(*
    Tests the free function F_AnyToUnionValue.
*)
{attribute 'call_after_init'}
FUNCTION_BLOCK FB_AnyToUnionValue_Test EXTENDS TcUnit.FB_TestSuite IMPLEMENTS TcUnit.I_RunnableTestSuite
VAR
    Assert : TcUnit.FB_Assert;
    
    aBit : BIT := 1; // Only structures and function blocks can have BIT defined
END_VAR

METHOD FB_init : BOOL
VAR_INPUT
	bInitRetains : BOOL; // if TRUE, the retain variables are initialized (warm start / cold start)
	bInCopyCode : BOOL;  // if TRUE, the instance afterwards gets moved into the copy code (online change)
END_VAR
SUPER^.RegisterTestSuite(THIS^);
END_METHOD

METHOD RunTests : TCUNIT.E_TestSuiteRunState
Test_BOOL();
Test_BIT();
Test_BYTE();
Test_WORD();
Test_DWORD();
Test_LWORD();
Test_SINT();
Test_INT();
Test_DINT();
Test_LINT();
Test_USINT();
Test_UINT();
Test_UDINT();
Test_ULINT();
Test_REAL();
Test_LREAL();
Test_STRING();
Test_STRING_2();
Test_WSTRING();
Test_TIME();
Test_DATE();
Test_DATE_AND_TIME();
Test_TIME_OF_DAY();
Test_LTIME();

RunTests := TCUNIT.E_TestSuiteRunState.FINISHED;
END_METHOD

METHOD PRIVATE Test_BIT
VAR
    result : U_ExpectedOrActual;
END_VAR
TEST('Test_BIT');

result := TcUnit.F_AnyToUnionValue(AnyValue := aBit);

Assert.AssertEquals(Expected := aBit,
                    Actual := result.bitExpectedOrActual,
                    Message := 'Values differ');
END_METHOD

METHOD PRIVATE Test_BOOL
VAR
    a : BOOL := TRUE;
    result : U_ExpectedOrActual;
END_VAR
TEST('Test_BOOL');

result := TcUnit.F_AnyToUnionValue(AnyValue := a);

Assert.AssertEquals(Expected := a,
                    Actual := result.boolExpectedOrActual,
                    Message := 'Values differ');
END_METHOD

METHOD PRIVATE Test_BYTE
VAR
    a : BYTE := 16#8A;
    result : U_ExpectedOrActual;
END_VAR
TEST('Test_BYTE');

result := TcUnit.F_AnyToUnionValue(AnyValue := a);

Assert.AssertEquals(Expected := a,
                    Actual := result.byteExpectedOrActual,
                    Message := 'Values differ');
END_METHOD

METHOD PRIVATE Test_DATE
VAR
    a : DATE := D#2106-02-05;
    result : U_ExpectedOrActual;
END_VAR
TEST('Test_DATE');

result := TcUnit.F_AnyToUnionValue(AnyValue := a);

Assert.AssertEquals(Expected := a,
                    Actual := result.dateExpectedOrActual,
                    Message := 'Values differ');
END_METHOD

METHOD PRIVATE Test_DATE_AND_TIME
VAR
    a : DATE_AND_TIME := DT#2106-02-06-06:28:15;
    result : U_ExpectedOrActual;
END_VAR
TEST('Test_DATE_AND_TIME');

result := TcUnit.F_AnyToUnionValue(AnyValue := a);

Assert.AssertEquals(Expected := a,
                    Actual := result.dateandtimeExpectedOrActual,
                    Message := 'Values differ');
END_METHOD

METHOD PRIVATE Test_DINT
VAR
    a : DINT := 143251;
    result : U_ExpectedOrActual;
END_VAR
TEST('Test_DINT');

result := TcUnit.F_AnyToUnionValue(AnyValue := a);

Assert.AssertEquals(Expected := a,
                    Actual := result.dintExpectedOrActual,
                    Message := 'Values differ');
END_METHOD

METHOD PRIVATE Test_DWORD
VAR
    a : DWORD := 16#3456CDEF;
    result : U_ExpectedOrActual;
END_VAR
TEST('Test_DWORD');

result := TcUnit.F_AnyToUnionValue(AnyValue := a);

Assert.AssertEquals(Expected := a,
                    Actual := result.dwordExpectedOrActual,
                    Message := 'Values differ');
END_METHOD

METHOD PRIVATE Test_INT
VAR
    a : INT := -32000;
    result : U_ExpectedOrActual;
END_VAR
TEST('Test_INT');

result := TcUnit.F_AnyToUnionValue(AnyValue := a);

Assert.AssertEquals(Expected := a,
                    Actual := result.intExpectedOrActual,
                    Message := 'Values differ');
END_METHOD

METHOD PRIVATE Test_LINT
VAR
    a : LINT := -31243145;
    result : U_ExpectedOrActual;
END_VAR
TEST('Test_LINT');

result := TcUnit.F_AnyToUnionValue(AnyValue := a);

Assert.AssertEquals(Expected := a,
                    Actual := result.lintExpectedOrActual,
                    Message := 'Values differ');
END_METHOD

METHOD PRIVATE Test_LREAL
VAR
    a : LREAL := 43123923124.745423;
    result : U_ExpectedOrActual;
END_VAR
TEST('Test_LREAL');

result := TcUnit.F_AnyToUnionValue(AnyValue := a);

Assert.AssertEquals(Expected := a,
                    Actual := result.lrealExpectedOrActual,
                    Message := 'Values differ');
END_METHOD

METHOD PRIVATE Test_LTIME
VAR
    a : LTIME := LTIME#213502D23H34M33S709MS551US615NS;
    result : U_ExpectedOrActual;
END_VAR
TEST('Test_LTIME');

result := TcUnit.F_AnyToUnionValue(AnyValue := a);

Assert.AssertEquals(Expected := a,
                    Actual := result.ltimeExpectedOrActual,
                    Message := 'Values differ');
END_METHOD

METHOD PRIVATE Test_LWORD
VAR
    a : LWORD := 16#456CDEF987654321;
    result : U_ExpectedOrActual;
END_VAR
TEST('Test_LWORD');

result := TcUnit.F_AnyToUnionValue(AnyValue := a);

Assert.AssertEquals(Expected := a,
                    Actual := result.lwordExpectedOrActual,
                    Message := 'Values differ');
END_METHOD

METHOD PRIVATE Test_REAL
VAR
    a : REAL := 431239.423;
    result : U_ExpectedOrActual;
END_VAR
TEST('Test_REAL');

result := TcUnit.F_AnyToUnionValue(AnyValue := a);

Assert.AssertEquals(Expected := a,
                    Actual := result.realExpectedOrActual,
                    Message := 'Values differ');
END_METHOD

METHOD PRIVATE Test_SINT
VAR
    a : SINT := 100;
    result : U_ExpectedOrActual;
END_VAR
TEST('Test_SINT');

result := TcUnit.F_AnyToUnionValue(AnyValue := a);

Assert.AssertEquals(Expected := a,
                    Actual := result.sintExpectedOrActual,
                    Message := 'Values differ');
END_METHOD

METHOD PRIVATE Test_STRING
VAR
    a : STRING := 'This is a random string';
    result : U_ExpectedOrActual;
END_VAR
TEST('Test_STRING');

result := TcUnit.F_AnyToUnionValue(AnyValue := a);

Assert.AssertEquals(Expected := a,
                    Actual := result.stringExpectedOrActual,
                    Message := 'Values differ');
END_METHOD

METHOD PRIVATE Test_STRING_2
VAR
    a : Tc2_System.T_MaxString := '8YNn5KOmPC4dAcpOBdLWnw4WkN126EwXsj65xeurG48gWBepinNaOIKeCVMtWNBSxQWPdtUYiAusDkjMLtQhDtiWbwvmoKcFwiUGDd7pOe0fd52J7hK60oaYAX6VWWmceLJX8utaDVrVzCGXafeZLeHl6jj5enfjg4tfb2WMEBdsBuG2iDKwzwhBLCPqXDnhe5HbemIbtZT7p62OEj2oDqiIYDD6tZdlhBCCelDBx6dbIp32wFm0TpRKsTiwkZ6'; // 255 characters
    result : U_ExpectedOrActual;
END_VAR
TEST('Test_STRING_2');

result := TcUnit.F_AnyToUnionValue(AnyValue := a);

Assert.AssertEquals(Expected := a,
                    Actual := result.stringExpectedOrActual,
                    Message := 'Values differ');
END_METHOD

METHOD PRIVATE Test_TIME
VAR
    a : TIME := T#15M20S;
    result : U_ExpectedOrActual;
END_VAR
TEST('Test_TIME');

result := TcUnit.F_AnyToUnionValue(AnyValue := a);

Assert.AssertEquals(Expected := a,
                    Actual := result.timeExpectedOrActual,
                    Message := 'Values differ');
END_METHOD

METHOD PRIVATE Test_TIME_OF_DAY
VAR
    a : TIME_OF_DAY := TOD#15:36:30.123;
    result : U_ExpectedOrActual;
END_VAR
TEST('Test_TIME_OF_DAY');

result := TcUnit.F_AnyToUnionValue(AnyValue := a);

Assert.AssertEquals(Expected := a,
                    Actual := result.timeofdayExpectedOrActual,
                    Message := 'Values differ');
END_METHOD

METHOD PRIVATE Test_UDINT
VAR
    a : UDINT := 2555;
    result : U_ExpectedOrActual;
END_VAR
TEST('Test_UDINT');

result := TcUnit.F_AnyToUnionValue(AnyValue := a);

Assert.AssertEquals(Expected := a,
                    Actual := result.udintExpectedOrActual,
                    Message := 'Values differ');
END_METHOD

METHOD PRIVATE Test_UINT
VAR
    a : UINT := 34523;
    result : U_ExpectedOrActual;
END_VAR
TEST('Test_UINT');

result := TcUnit.F_AnyToUnionValue(AnyValue := a);

Assert.AssertEquals(Expected := a,
                    Actual := result.uintExpectedOrActual,
                    Message := 'Values differ');
END_METHOD

METHOD PRIVATE Test_ULINT
VAR
    a : ULINT := 25555423;
    result : U_ExpectedOrActual;
END_VAR
TEST('TEST_ULINT');

result := TcUnit.F_AnyToUnionValue(AnyValue := a);

Assert.AssertEquals(Expected := a,
                    Actual := result.ulintExpectedOrActual,
                    Message := 'Values differ');
END_METHOD

METHOD PRIVATE Test_USINT
VAR
    a : USINT := 255;
    result : U_ExpectedOrActual;
END_VAR
TEST('Test_USINT');

result := TcUnit.F_AnyToUnionValue(AnyValue := a);

Assert.AssertEquals(Expected := a,
                    Actual := result.usintExpectedOrActual,
                    Message := 'Values differ');
END_METHOD

METHOD PRIVATE Test_WORD
VAR
    a : WORD := 16#ABCD;
    result : U_ExpectedOrActual;
END_VAR
TEST('Test_WORD');

result := TcUnit.F_AnyToUnionValue(AnyValue := a);

Assert.AssertEquals(Expected := a,
                    Actual := result.wordExpectedOrActual,
                    Message := 'Values differ');
END_METHOD

METHOD PRIVATE Test_WSTRING
VAR
    a : WSTRING := "This is a random string";
    result : U_ExpectedOrActual;
END_VAR
TEST('Test_WSTRING');

result := TcUnit.F_AnyToUnionValue(AnyValue := a);

Assert.AssertEquals(Expected := a,
                    Actual := result.wstringExpectedOrActual,
                    Message := 'Values differ');
END_METHOD

END_FUNCTION_BLOCK

(* stored: Version 1.1.0.1, ProductVersion 3.1.4022.16
   POU FB_AnyToUnionValue_Test: Id {0cc46357-158c-41b7-afc0-2c79ec82f0f6}, SpecialFunc None
   Method FB_init: Id {0485650c-1465-4486-a734-95b061eb38ae}
   Method RunTests: Id {7fda42d2-1918-424a-ba0f-a586afc09af2}
   Method Test_BIT: Id {2bab70c5-093e-48a7-94e6-ae7f2bb2e7b3}
   Method Test_BOOL: Id {48f55beb-9fc1-4336-8784-72fc7eda80de}
   Method Test_BYTE: Id {226781dc-3660-487a-bcbd-00cc36750e0e}
   Method Test_DATE: Id {84a5fde1-b357-4804-bf01-5c83bfeb54b3}
   Method Test_DATE_AND_TIME: Id {76b46507-8743-481c-8853-3b45d1544ad5}
   Method Test_DINT: Id {c81a9536-5ff4-4424-9f7e-1d8c5133b5e3}
   Method Test_DWORD: Id {e6dfcf37-a491-45b2-9543-b7fdd8847283}
   Method Test_INT: Id {77ff5bf1-1822-4366-a4ee-34a185c0d47e}
   Method Test_LINT: Id {d2a7cc80-d43e-4823-a346-11defa0d180f}
   Method Test_LREAL: Id {af2fee48-9d46-49ec-9fe0-6a046d6c2f7d}
   Method Test_LTIME: Id {1affac86-d501-40a0-99f5-4eeb9cd389fd}
   Method Test_LWORD: Id {f0464dd4-9a3f-4fed-bf6c-84c05edc34ab}
   Method Test_REAL: Id {5ff5264d-4661-4dc4-8889-01d457341535}
   Method Test_SINT: Id {fd59d157-95aa-462e-812a-26f74d790e8c}
   Method Test_STRING: Id {825e7694-a502-4c32-9d34-807560d3aa4c}
   Method Test_STRING_2: Id {1e075eec-d55a-483a-976e-656d4a8d5ac3}
   Method Test_TIME: Id {e7b3c2aa-6660-47ce-9edf-58924221789c}
   Method Test_TIME_OF_DAY: Id {55ccbe56-fcd0-4e7f-8497-d0c19c60ad6a}
   Method Test_UDINT: Id {2ae444f0-9149-4c01-b7ad-2fdcab7bba7c}
   Method Test_UINT: Id {3309739e-f1a1-45d7-928b-c636d1592c1c}
   Method Test_ULINT: Id {5e5e97df-5e62-40a2-b054-3ba7c91cef70}
   Method Test_USINT: Id {ef948bb4-ae4e-47a7-b963-d71ce86c9997}
   Method Test_WORD: Id {3859891c-ade4-48ca-89f8-da9a77a2ccbb}
   Method Test_WSTRING: Id {cd24edfa-28c7-4bf7-ad9e-262f073a3ddf} *)
